INTERFACE I_KeyValueCollectionChangedEvent EXTENDS I_Event

PROPERTY PUBLIC Target : I_KeyValueCollection
GET
END_GET
END_PROPERTY

END_INTERFACE

(* stored: Version 1.1.0.1, ProductVersion 3.1.4024.12
   Itf I_KeyValueCollectionChangedEvent: Id {5602f461-bede-0bfe-1ff5-4565325aa1c3}
   Property Target: Id {69331e0a-b84f-07af-309d-d43fba57bc5e}
   Get Get: Id {eb53bf45-35ec-0c26-0739-9c140879e9a0} *)
